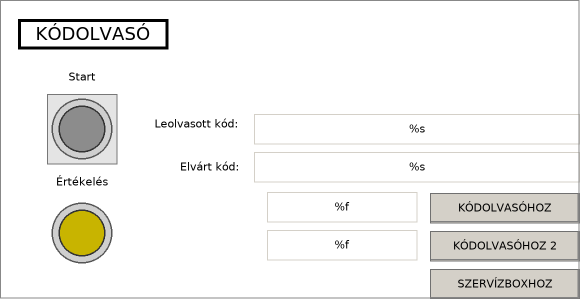
VISUALIZATION Kodolvaso  // 580x299
    PushSwitch (47,94 70x70), variable: ZEBRASCANNER.bStartSend, behaviour: TOGGLE, style: Switch-PushSwitch-Gray
    Lamp1 (47,198 70x70), variable: GVL.bMarkingOK, style: Lamp-Lamp1-Yellow
    Textfield (254,114 326x30), "%s", text variable: ZEBRASCANNER.sReceivedString255
    Label (48,67 68x20), "Start"
    Label (48,172 68x20), "Értékelés"
    Label (149,114 92x20), "Leolvasott kód:"
    Label (150,157 92x20), "Elvárt kód:"
    Textfield (254,152 326x30), "%s", text variable: ZEBRASCANNER.sExpectedString
    RoundedRectangle (18,19 150x30)
    Label (18,19 150x30), "KÓDOLVASÓ"
    Textfield (267,192 150x30), "%f", text variable: GVL.lrKodolvasasPosition
        OnMouseClick: write the text variable via VisuDialogs.Numpad, min -10000, max -1
    Button (430,193 150x30), "KÓDOLVASÓHOZ"
        OnMouseUp: execute { PISTITENGELY.lrPistiPosition:=GVL.lrKodolvasasPosition; PISTITENGELY.sPistiAxisCommand:='MOVE'; }
    Button (430,269 150x30), "SZERVÍZBOXHOZ"
        OnMouseUp: execute { PISTITENGELY.lrPistiPosition:=GVL.lrPtSzervizbox; PISTITENGELY.sPistiAxisCommand:='MOVE'; }
    Textfield (267,230 150x30), "%f", text variable: GVL.lrKodolvasasPosition2
        OnMouseClick: write the text variable via VisuDialogs.Numpad, min -10000, max -1
    Button (430,231 150x30), "KÓDOLVASÓHOZ 2"
        OnMouseUp: execute { PISTITENGELY.lrPistiPosition:=GVL.lrKodolvasasPosition2; PISTITENGELY.sPistiAxisCommand:='MOVE'; }
END_VISUALIZATION

(* stored: Version 1.1.0.1, ProductVersion 3.1.4024.11
   Visu Kodolvaso: Id {0bc0c138-2a9e-4c11-868e-cabb17ce1e26} *)
